TYPE ST_CoaxVisionCommunicationConfig :
STRUCT
    // PLC发出测量请求后等待Python Vision Service返回对应ResultId的最长时间。
    tResultTimeout : TIME;
END_STRUCT
END_TYPE

(* stored: Version 1.1.0.1, ProductVersion 3.1.4026.20
   DUT ST_CoaxVisionCommunicationConfig: Id {A2867EDC-3B38-49D8-B0BA-2776085C0D02} *)
